FUNCTION_BLOCK "_UtilitiesFB"
{ S7_Optimized_Access := 'TRUE' }
VERSION : 0.1
   VAR_INPUT
      CPUSytemMemoryBits { ExternalAccessible := 'False'; ExternalVisible := 'False'; ExternalWritable := 'False'; } : Byte;   // Address of system memory byte
      CPUClockMemoryBits { ExternalAccessible := 'False'; ExternalVisible := 'False'; ExternalWritable := 'False'; } : Byte;   // Address of clock memory byte
      StartupDelaySP { ExternalAccessible := 'False'; ExternalVisible := 'False'; ExternalWritable := 'False'; } : Time;   // Delay before startup delay bit turned on
   END_VAR

   VAR
      AlwaysOn { ExternalAccessible := 'False'; ExternalVisible := 'False'; ExternalWritable := 'False'; } : Bool;   // Bit always TRUE
      AlwaysTrue { ExternalAccessible := 'False'; ExternalVisible := 'False'; ExternalWritable := 'False'; } : Bool;   // Bit always TRUE
      AlwaysOff { ExternalAccessible := 'False'; ExternalVisible := 'False'; ExternalWritable := 'False'; } : Bool;   // Bit always FALSE
      AlwaysFalse { ExternalAccessible := 'False'; ExternalVisible := 'False'; ExternalWritable := 'False'; } : Bool;   // Bit always FALSE
      FirstScan { ExternalAccessible := 'False'; ExternalVisible := 'False'; ExternalWritable := 'False'; } : Bool;   // Bit TRUE for only the first scan of the PLC
      StartupDelayDn { ExternalAccessible := 'False'; ExternalVisible := 'False'; ExternalWritable := 'False'; } : Bool;   // Bit initially FALSE, turning TRUE after preset delay
      StartupDelayTmr { ExternalAccessible := 'False'; ExternalVisible := 'False'; ExternalWritable := 'False'; OriginalPartName := 'IEC_TIMER'; LibVersion := '1.0'} : IEC_TIMER;
      Square_100ms { ExternalAccessible := 'False'; ExternalVisible := 'False'; ExternalWritable := 'False'; } : Bool;   // Bit FALSE/TRUE based on square wave (100 ms frequency)
      Square_100msONS { ExternalAccessible := 'False'; ExternalVisible := 'False'; ExternalWritable := 'False'; } : Bool;
      Pulse_100ms { ExternalAccessible := 'False'; ExternalVisible := 'False'; ExternalWritable := 'False'; } : Bool;   // Bit TRUE every 100 ms for one PLC scan
      Square_200ms { ExternalAccessible := 'False'; ExternalVisible := 'False'; ExternalWritable := 'False'; } : Bool;   // Bit FALSE/TRUE based on square wave (200 ms frequency)
      Square_200msONS { ExternalAccessible := 'False'; ExternalVisible := 'False'; ExternalWritable := 'False'; } : Bool;
      Pulse_200ms { ExternalAccessible := 'False'; ExternalVisible := 'False'; ExternalWritable := 'False'; } : Bool;   // Bit TRUE every 200 ms for one PLC scan
      Square_400ms { ExternalAccessible := 'False'; ExternalVisible := 'False'; ExternalWritable := 'False'; } : Bool;   // Bit FALSE/TRUE based on square wave (400 ms frequency)
      Square_400msONS { ExternalAccessible := 'False'; ExternalVisible := 'False'; ExternalWritable := 'False'; } : Bool;
      Pulse_400ms { ExternalAccessible := 'False'; ExternalVisible := 'False'; ExternalWritable := 'False'; } : Bool;   // Bit TRUE every 400 ms for one PLC scan
      Square_500ms { ExternalAccessible := 'False'; ExternalVisible := 'False'; ExternalWritable := 'False'; } : Bool;   // Bit FALSE/TRUE based on square wave (500 ms frequency)
      Square_500msONS { ExternalAccessible := 'False'; ExternalVisible := 'False'; ExternalWritable := 'False'; } : Bool;
      Pulse_500ms { ExternalAccessible := 'False'; ExternalVisible := 'False'; ExternalWritable := 'False'; } : Bool;   // Bit TRUE every 500 ms for one PLC scan
      Square_800ms { ExternalAccessible := 'False'; ExternalVisible := 'False'; ExternalWritable := 'False'; } : Bool;   // Bit FALSE/TRUE based on square wave (800 ms frequency)
      Square_800msONS { ExternalAccessible := 'False'; ExternalVisible := 'False'; ExternalWritable := 'False'; } : Bool;
      Pulse_800ms { ExternalAccessible := 'False'; ExternalVisible := 'False'; ExternalWritable := 'False'; } : Bool;   // Bit TRUE every 800 ms for one PLC scan
      Square_1s { ExternalAccessible := 'False'; ExternalVisible := 'False'; ExternalWritable := 'False'; } : Bool;   // Bit FALSE/TRUE based on square wave (1 s frequency)
      Square_1sONS { ExternalAccessible := 'False'; ExternalVisible := 'False'; ExternalWritable := 'False'; } : Bool;
      Pulse_1s { ExternalAccessible := 'False'; ExternalVisible := 'False'; ExternalWritable := 'False'; } : Bool;   // Bit TRUE every 1 s for one PLC scan
      Square_1600ms { ExternalAccessible := 'False'; ExternalVisible := 'False'; ExternalWritable := 'False'; } : Bool;   // Bit FALSE/TRUE based on square wave (1600 ms frequency)
      Square_1600msONS { ExternalAccessible := 'False'; ExternalVisible := 'False'; ExternalWritable := 'False'; } : Bool;
      Pulse_1600ms { ExternalAccessible := 'False'; ExternalVisible := 'False'; ExternalWritable := 'False'; } : Bool;   // Bit TRUE every 1600 ms for one PLC scan
      Square_2s { ExternalAccessible := 'False'; ExternalVisible := 'False'; ExternalWritable := 'False'; } : Bool;   // Bit FALSE/TRUE based on square wave (2 s frequency)
      Square_2sONS { ExternalAccessible := 'False'; ExternalVisible := 'False'; ExternalWritable := 'False'; } : Bool;
      Pulse_2s { ExternalAccessible := 'False'; ExternalVisible := 'False'; ExternalWritable := 'False'; } : Bool;   // Bit TRUE every 2 s for one PLC scan
      TestInProgress { ExternalAccessible := 'False'; ExternalVisible := 'False'; ExternalWritable := 'False'; } : Bool;   // Indicates which caller FC is used
      EPICS_Device_calls_precessed { ExternalAccessible := 'False'; ExternalVisible := 'False'; ExternalWritable := 'False'; } : Bool;   // Indicates which caller FC is used
   END_VAR

BEGIN
	//This block provides standard "Utilities" tags that can be used in the rest OF the PLC code such
	//as:
	//* Always On
	//* Always Off
	//* Startup Delay
	//* Pulses (different frequences)
	//* etc.

	//When using This block in your program, name the instance DB "Utilities" AND THEN you will be able TO use tags like "Utilities.AlwaysOn" in the rest OF your program.

	//This block relies On information provided BY the CPU. This needs TO be enabled in the CPU hardware configuration under System AND Clock Memory.
	//Enable both functions AND pick memory bytes you'd like TO use (defauls are %MB1 AND %MB0 respectively).
	//THEN connect the selected Byte TO the inputs OF This block.
	//

	//Bit TRUE for only the first scan of the PLC
	#FirstScan := #CPUSytemMemoryBits.%X0;

	//Bit always TRUE
	#AlwaysOn := #CPUSytemMemoryBits.%X2;
	#AlwaysTrue := #CPUSytemMemoryBits.%X2;

	//Bit always FALSE
	#AlwaysOff := #CPUSytemMemoryBits.%X3;
	#AlwaysFalse := #CPUSytemMemoryBits.%X3;

	//Bit initially FALSE, turning TRUE after preset delay
	#StartupDelayTmr.TON(IN := #AlwaysTrue,
	                     PT := #StartupDelaySP,
	                     Q => #StartupDelayDn);

	//Bit TRUE every 100 ms FOR one PLC scan
	#Square_100ms := #CPUClockMemoryBits.%X0;
	"UTIL_P_TRIG"("i_Input Bit" := #Square_100ms,
	              "iq_Trigger Bit" := #Square_100msONS,
	              "iq_Pulse Bit" := #Pulse_100ms);

	//Bit TRUE every 200 ms FOR one PLC scan
	#Square_200ms := #CPUClockMemoryBits.%X1;
	"UTIL_P_TRIG"("i_Input Bit" := #Square_200ms,
	              "iq_Trigger Bit" := #Square_200msONS,
	              "iq_Pulse Bit" := #Pulse_200ms);

	//Bit TRUE every 400 ms FOR one PLC scan
	#Square_400ms := #CPUClockMemoryBits.%X2;
	"UTIL_P_TRIG"("i_Input Bit" := #Square_400ms,
	              "iq_Trigger Bit" := #Square_400msONS,
	              "iq_Pulse Bit" := #Pulse_400ms);

	//Bit TRUE every 500 ms FOR one PLC scan
	#Square_500ms := #CPUClockMemoryBits.%X3;
	"UTIL_P_TRIG"("i_Input Bit" := #Square_500ms,
	              "iq_Trigger Bit" := #Square_500msONS,
	              "iq_Pulse Bit" := #Pulse_500ms);

	//Bit TRUE every 800 ms FOR one PLC scan
	#Square_800ms := #CPUClockMemoryBits.%X4;
	"UTIL_P_TRIG"("i_Input Bit" := #Square_800ms,
	              "iq_Trigger Bit" := #Square_800msONS,
	              "iq_Pulse Bit" := #Pulse_800ms);

	//Bit TRUE every 1 s FOR one PLC scan
	#Square_1s := #CPUClockMemoryBits.%X5;
	"UTIL_P_TRIG"("i_Input Bit" := #Square_1s,
	              "iq_Trigger Bit" := #Square_1sONS,
	              "iq_Pulse Bit" := #Pulse_1s);

	//Bit TRUE every 1600 ms FOR one PLC scan
	#Square_1600ms := #CPUClockMemoryBits.%X6;
	"UTIL_P_TRIG"("i_Input Bit" := #Square_1600ms,
	              "iq_Trigger Bit" := #Square_1600msONS,
	              "iq_Pulse Bit" := #Pulse_1600ms);

	//Bit TRUE every 2s FOR one PLC scan
	#Square_2s := #CPUClockMemoryBits.%X7;
	"UTIL_P_TRIG"("i_Input Bit" := #Square_2s,
	              "iq_Trigger Bit" := #Square_2sONS,
	              "iq_Pulse Bit" := #Pulse_2s);

END_FUNCTION_BLOCK
DATA_BLOCK "Utilities"
{ S7_Optimized_Access := 'TRUE' }
VERSION : 0.1
NON_RETAIN
"_UtilitiesFB"

BEGIN

END_DATA_BLOCK
FUNCTION_BLOCK "DEVTYPE_ISRC_LEBT_BDump"
{ S7_Optimized_Access := 'TRUE' }
VERSION : 1.0
   VAR_INPUT
      "WtrFlowOK" { ExternalAccessible := 'True'; ExternalVisible := 'False'; ExternalWritable := 'False'; } : BOOL;   //EPICS Status variable: WtrFlowOK
   EPICSToPLCLength { ExternalAccessible := 'False'; ExternalVisible := 'False'; ExternalWritable := 'False'; } : Int;   // Length of device command register array (in words)
   EPICSToPLCDataBlockOffset { ExternalAccessible := 'False'; ExternalVisible := 'False'; ExternalWritable := 'False'; } : Int;   // Offset in EPICS->PLC comms block where this device data resides (in words)
   EPICSToPLCParametersStart { ExternalAccessible := 'False'; ExternalVisible := 'False'; ExternalWritable := 'False'; } : Int;   // The border offset between the Command and the Parameter area
   PLCToEPICSLength { ExternalAccessible := 'False'; ExternalVisible := 'False'; ExternalWritable := 'False'; } : Int;   // Length of device status register array (in words)
   PLCToEPICSDataBlockOffset { ExternalAccessible := 'False'; ExternalVisible := 'False'; ExternalWritable := 'False'; } : Int;   // Offset in PLC->EPICS comms block where this device data resides (in words)
   END_VAR
   VAR_OUTPUT
      DEVICE_PARAM_OK { ExternalAccessible := 'False'; ExternalVisible := 'False'; ExternalWritable := 'False'; } : Bool;
   END_VAR
   VAR_IN_OUT
   END_VAR
   Var DB_SPECIFIC
      MyWord { ExternalAccessible := 'False'; ExternalVisible := 'False'; ExternalWritable := 'False'; } : Word;
      MyBytesinWord { ExternalAccessible := 'False'; ExternalVisible := 'False'; ExternalWritable := 'False'; } AT MyWord : Array[0..1] of Byte;
      MyBoolsinWord { ExternalAccessible := 'False'; ExternalVisible := 'False'; ExternalWritable := 'False'; } AT MyWord : Array[0..15] of Bool;
      MyDInt { ExternalAccessible := 'False'; ExternalVisible := 'False'; ExternalWritable := 'False'; } : DInt;
      MyWordsinDint { ExternalAccessible := 'False'; ExternalVisible := 'False'; ExternalWritable := 'False'; } AT MyDInt : Array[0..1] of Word;
      MyReal { ExternalAccessible := 'False'; ExternalVisible := 'False'; ExternalWritable := 'False'; } : Real;
      MyWordsinReal { ExternalAccessible := 'False'; ExternalVisible := 'False'; ExternalWritable := 'False'; } AT MyReal : Array[0..1] of Word;
      MyInt { ExternalAccessible := 'False'; ExternalVisible := 'False'; ExternalWritable := 'False'; } : Int;
      MyWordinInt { ExternalAccessible := 'False'; ExternalVisible := 'False'; ExternalWritable := 'False'; } AT MyInt : Word;
      MyDWord { ExternalAccessible := 'False'; ExternalVisible := 'False'; ExternalWritable := 'False'; } : DWord;
      MyWordsinDWord { ExternalAccessible := 'False'; ExternalVisible := 'False'; ExternalWritable := 'False'; } AT MyDWord : Array[0..1] of Word;
      MyTime { ExternalAccessible := 'False'; ExternalVisible := 'False'; ExternalWritable := 'False'; } : Time;
      MyWordsinTime { ExternalAccessible := 'False'; ExternalVisible := 'False'; ExternalWritable := 'False'; } AT MyTime : Array[0..1] of Word;
      MyString { ExternalAccessible := 'False'; ExternalVisible := 'False'; ExternalWritable := 'False'; } : String[40];
      MyWordsinString { ExternalAccessible := 'False'; ExternalVisible := 'False'; ExternalWritable := 'False'; } AT MyString : Array[0..20] of Word;
   END_VAR
   VAR_TEMP
      HashModbus : DInt;
      HashIFA : DInt;
      HashTIAMap : DInt;
      i : Int;
   END_VAR
    //Author: Miklos Boros (miklos.boros@esss.se), Copyrigth 2017-2019 by European Spallation Source, Lund
    //This block was generated by PLCFactory, please don't change it MANUALLY!
    //Input File Name: ISrc-010_Ctrl-PLC-01-template-IFA-20191106135317.ifa
    //Generated: 20191106135317
    //According to HASH: 1347332123
    //Device type: ISRC_LEBT_BDump
    //Description: This function does the variable mapping for a device. All device-variable will be linked to an interface variable defined in this block.

    //********************************************
    //****************HASH check******************
    //********************************************


    #MyWordsinDint[0] := "EPICSToPLC"."Word"[0];
    #MyWordsinDint[1] := "EPICSToPLC"."Word"[1];
    #HashModbus := #MyDInt; //Hash from EPICS/ModbusTCP

    #HashIFA := 1347332123; //Hash from Interface Factory as a constant

    #MyWordsinDint[0] := "PLCToEPICS"."Word"[0];
    #MyWordsinDint[1] := "PLCToEPICS"."Word"[1];
    #HashTIAMap := #MyDInt; //Hash from PLCFactory TIA Map


    IF ((#HashIFA = #HashModbus) AND (#HashModbus = #HashTIAMap)) THEN //Check CRCs
        #DEVICE_PARAM_OK := TRUE;
       //###########################  LEBT Beam Dump  ##############################
       //###########################
       //STATUS BLOCK
       //###########################

    //********************************************
    //*************STATUS VARIABLES***************
    //********************************************


       #MyWord := W#0;
       #MyBoolsinWord[8] := #"WtrFlowOK";    //EPICSName: WtrFlowOK
       "PLCToEPICS"."Word"[#PLCToEPICSDataBlockOffset + 0] := #MyWord;
    Else
       #DEVICE_PARAM_OK := FALSE; //Invalid Hash
    END_IF;
END_FUNCTION_BLOCK
FUNCTION_BLOCK "DEVTYPE_ISRC_LEBT_CHOP"
{ S7_Optimized_Access := 'TRUE' }
VERSION : 1.0
   VAR_INPUT
      "PwrSysOK" { ExternalAccessible := 'True'; ExternalVisible := 'False'; ExternalWritable := 'False'; } : BOOL;   //EPICS Status variable: PwrSysOK
      "ChopVoltAlarmR" { ExternalAccessible := 'True'; ExternalVisible := 'False'; ExternalWritable := 'False'; } : BOOL;   //EPICS Status variable: ChopVoltAlarmR
      "WtrFlowOK" { ExternalAccessible := 'True'; ExternalVisible := 'False'; ExternalWritable := 'False'; } : BOOL;   //EPICS Status variable: WtrFlowOK
      "HVEnCmdRB" { ExternalAccessible := 'True'; ExternalVisible := 'False'; ExternalWritable := 'False'; } : BOOL;   //EPICS Status variable: HVEnCmdRB
   EPICSToPLCLength { ExternalAccessible := 'False'; ExternalVisible := 'False'; ExternalWritable := 'False'; } : Int;   // Length of device command register array (in words)
   EPICSToPLCDataBlockOffset { ExternalAccessible := 'False'; ExternalVisible := 'False'; ExternalWritable := 'False'; } : Int;   // Offset in EPICS->PLC comms block where this device data resides (in words)
   EPICSToPLCParametersStart { ExternalAccessible := 'False'; ExternalVisible := 'False'; ExternalWritable := 'False'; } : Int;   // The border offset between the Command and the Parameter area
   PLCToEPICSLength { ExternalAccessible := 'False'; ExternalVisible := 'False'; ExternalWritable := 'False'; } : Int;   // Length of device status register array (in words)
   PLCToEPICSDataBlockOffset { ExternalAccessible := 'False'; ExternalVisible := 'False'; ExternalWritable := 'False'; } : Int;   // Offset in PLC->EPICS comms block where this device data resides (in words)
   END_VAR
   VAR_OUTPUT
      "HVEnOnCmd" { ExternalAccessible := 'True'; ExternalVisible := 'False'; ExternalWritable := 'False'; } : BOOL;   //EPICS Command variable: HVEnOnCmd
      "HVEnOffCmd" { ExternalAccessible := 'True'; ExternalVisible := 'False'; ExternalWritable := 'False'; } : BOOL;   //EPICS Command variable: HVEnOffCmd
      DEVICE_PARAM_OK { ExternalAccessible := 'False'; ExternalVisible := 'False'; ExternalWritable := 'False'; } : Bool;
   END_VAR
   VAR_IN_OUT
   END_VAR
   Var DB_SPECIFIC
      MyWord { ExternalAccessible := 'False'; ExternalVisible := 'False'; ExternalWritable := 'False'; } : Word;
      MyBytesinWord { ExternalAccessible := 'False'; ExternalVisible := 'False'; ExternalWritable := 'False'; } AT MyWord : Array[0..1] of Byte;
      MyBoolsinWord { ExternalAccessible := 'False'; ExternalVisible := 'False'; ExternalWritable := 'False'; } AT MyWord : Array[0..15] of Bool;
      MyDInt { ExternalAccessible := 'False'; ExternalVisible := 'False'; ExternalWritable := 'False'; } : DInt;
      MyWordsinDint { ExternalAccessible := 'False'; ExternalVisible := 'False'; ExternalWritable := 'False'; } AT MyDInt : Array[0..1] of Word;
      MyReal { ExternalAccessible := 'False'; ExternalVisible := 'False'; ExternalWritable := 'False'; } : Real;
      MyWordsinReal { ExternalAccessible := 'False'; ExternalVisible := 'False'; ExternalWritable := 'False'; } AT MyReal : Array[0..1] of Word;
      MyInt { ExternalAccessible := 'False'; ExternalVisible := 'False'; ExternalWritable := 'False'; } : Int;
      MyWordinInt { ExternalAccessible := 'False'; ExternalVisible := 'False'; ExternalWritable := 'False'; } AT MyInt : Word;
      MyDWord { ExternalAccessible := 'False'; ExternalVisible := 'False'; ExternalWritable := 'False'; } : DWord;
      MyWordsinDWord { ExternalAccessible := 'False'; ExternalVisible := 'False'; ExternalWritable := 'False'; } AT MyDWord : Array[0..1] of Word;
      MyTime { ExternalAccessible := 'False'; ExternalVisible := 'False'; ExternalWritable := 'False'; } : Time;
      MyWordsinTime { ExternalAccessible := 'False'; ExternalVisible := 'False'; ExternalWritable := 'False'; } AT MyTime : Array[0..1] of Word;
      MyString { ExternalAccessible := 'False'; ExternalVisible := 'False'; ExternalWritable := 'False'; } : String[40];
      MyWordsinString { ExternalAccessible := 'False'; ExternalVisible := 'False'; ExternalWritable := 'False'; } AT MyString : Array[0..20] of Word;
   END_VAR
   VAR_TEMP
      HashModbus : DInt;
      HashIFA : DInt;
      HashTIAMap : DInt;
      i : Int;
   END_VAR
    //Author: Miklos Boros (miklos.boros@esss.se), Copyrigth 2017-2019 by European Spallation Source, Lund
    //This block was generated by PLCFactory, please don't change it MANUALLY!
    //Input File Name: ISrc-010_Ctrl-PLC-01-template-IFA-20191106135317.ifa
    //Generated: 20191106135317
    //According to HASH: 1347332123
    //Device type: ISRC_LEBT_CHOP
    //Description: This function does the variable mapping for a device. All device-variable will be linked to an interface variable defined in this block.

    //********************************************
    //****************HASH check******************
    //********************************************


    #MyWordsinDint[0] := "EPICSToPLC"."Word"[0];
    #MyWordsinDint[1] := "EPICSToPLC"."Word"[1];
    #HashModbus := #MyDInt; //Hash from EPICS/ModbusTCP

    #HashIFA := 1347332123; //Hash from Interface Factory as a constant

    #MyWordsinDint[0] := "PLCToEPICS"."Word"[0];
    #MyWordsinDint[1] := "PLCToEPICS"."Word"[1];
    #HashTIAMap := #MyDInt; //Hash from PLCFactory TIA Map


    IF ((#HashIFA = #HashModbus) AND (#HashModbus = #HashTIAMap)) THEN //Check CRCs
        #DEVICE_PARAM_OK := TRUE;
       //###########################  LEBT Chopper  ##############################
       //###########################
       //STATUS BLOCK
       //###########################

    //********************************************
    //*************STATUS VARIABLES***************
    //********************************************


       #MyWord := W#0;
       #MyBoolsinWord[8] := #"PwrSysOK";    //EPICSName: PwrSysOK
       #MyBoolsinWord[9] := #"ChopVoltAlarmR";    //EPICSName: ChopVoltAlarmR
       #MyBoolsinWord[10] := #"WtrFlowOK";    //EPICSName: WtrFlowOK
       #MyBoolsinWord[11] := #"HVEnCmdRB";    //EPICSName: HVEnCmdRB
       "PLCToEPICS"."Word"[#PLCToEPICSDataBlockOffset + 0] := #MyWord;

    //********************************************
    //*************COMMAND VARIABLES**************
    //********************************************


       #MyWord := "EPICSToPLC"."Word"[#EPICSToPLCDataBlockOffset + 0];
       IF (NOT "Utilities".TestInProgress) THEN
       	"EPICSToPLC"."Word"[#EPICSToPLCDataBlockOffset + 0] := 0;
       END_IF;
       #"HVEnOnCmd" := #MyBoolsinWord[8];    //EPICSName: HVEnOnCmd
       #"HVEnOffCmd" := #MyBoolsinWord[9];    //EPICSName: HVEnOffCmd
    Else
       #DEVICE_PARAM_OK := FALSE; //Invalid Hash
    END_IF;
END_FUNCTION_BLOCK
FUNCTION_BLOCK "DEVTYPE_ISRC_LEBT_COIL_SOLENOID"
{ S7_Optimized_Access := 'TRUE' }
VERSION : 1.0
   VAR_INPUT
      "WtrFlowOK" { ExternalAccessible := 'True'; ExternalVisible := 'False'; ExternalWritable := 'False'; } : BOOL;   //EPICS Status variable: WtrFlowOK
      "WtrTempOK" { ExternalAccessible := 'True'; ExternalVisible := 'False'; ExternalWritable := 'False'; } : BOOL;   //EPICS Status variable: WtrTempOK
   EPICSToPLCLength { ExternalAccessible := 'False'; ExternalVisible := 'False'; ExternalWritable := 'False'; } : Int;   // Length of device command register array (in words)
   EPICSToPLCDataBlockOffset { ExternalAccessible := 'False'; ExternalVisible := 'False'; ExternalWritable := 'False'; } : Int;   // Offset in EPICS->PLC comms block where this device data resides (in words)
   EPICSToPLCParametersStart { ExternalAccessible := 'False'; ExternalVisible := 'False'; ExternalWritable := 'False'; } : Int;   // The border offset between the Command and the Parameter area
   PLCToEPICSLength { ExternalAccessible := 'False'; ExternalVisible := 'False'; ExternalWritable := 'False'; } : Int;   // Length of device status register array (in words)
   PLCToEPICSDataBlockOffset { ExternalAccessible := 'False'; ExternalVisible := 'False'; ExternalWritable := 'False'; } : Int;   // Offset in PLC->EPICS comms block where this device data resides (in words)
   END_VAR
   VAR_OUTPUT
      DEVICE_PARAM_OK { ExternalAccessible := 'False'; ExternalVisible := 'False'; ExternalWritable := 'False'; } : Bool;
   END_VAR
   VAR_IN_OUT
   END_VAR
   Var DB_SPECIFIC
      MyWord { ExternalAccessible := 'False'; ExternalVisible := 'False'; ExternalWritable := 'False'; } : Word;
      MyBytesinWord { ExternalAccessible := 'False'; ExternalVisible := 'False'; ExternalWritable := 'False'; } AT MyWord : Array[0..1] of Byte;
      MyBoolsinWord { ExternalAccessible := 'False'; ExternalVisible := 'False'; ExternalWritable := 'False'; } AT MyWord : Array[0..15] of Bool;
      MyDInt { ExternalAccessible := 'False'; ExternalVisible := 'False'; ExternalWritable := 'False'; } : DInt;
      MyWordsinDint { ExternalAccessible := 'False'; ExternalVisible := 'False'; ExternalWritable := 'False'; } AT MyDInt : Array[0..1] of Word;
      MyReal { ExternalAccessible := 'False'; ExternalVisible := 'False'; ExternalWritable := 'False'; } : Real;
      MyWordsinReal { ExternalAccessible := 'False'; ExternalVisible := 'False'; ExternalWritable := 'False'; } AT MyReal : Array[0..1] of Word;
      MyInt { ExternalAccessible := 'False'; ExternalVisible := 'False'; ExternalWritable := 'False'; } : Int;
      MyWordinInt { ExternalAccessible := 'False'; ExternalVisible := 'False'; ExternalWritable := 'False'; } AT MyInt : Word;
      MyDWord { ExternalAccessible := 'False'; ExternalVisible := 'False'; ExternalWritable := 'False'; } : DWord;
      MyWordsinDWord { ExternalAccessible := 'False'; ExternalVisible := 'False'; ExternalWritable := 'False'; } AT MyDWord : Array[0..1] of Word;
      MyTime { ExternalAccessible := 'False'; ExternalVisible := 'False'; ExternalWritable := 'False'; } : Time;
      MyWordsinTime { ExternalAccessible := 'False'; ExternalVisible := 'False'; ExternalWritable := 'False'; } AT MyTime : Array[0..1] of Word;
      MyString { ExternalAccessible := 'False'; ExternalVisible := 'False'; ExternalWritable := 'False'; } : String[40];
      MyWordsinString { ExternalAccessible := 'False'; ExternalVisible := 'False'; ExternalWritable := 'False'; } AT MyString : Array[0..20] of Word;
   END_VAR
   VAR_TEMP
      HashModbus : DInt;
      HashIFA : DInt;
      HashTIAMap : DInt;
      i : Int;
   END_VAR
    //Author: Miklos Boros (miklos.boros@esss.se), Copyrigth 2017-2019 by European Spallation Source, Lund
    //This block was generated by PLCFactory, please don't change it MANUALLY!
    //Input File Name: ISrc-010_Ctrl-PLC-01-template-IFA-20191106135317.ifa
    //Generated: 20191106135317
    //According to HASH: 1347332123
    //Device type: ISRC_LEBT_COIL_SOLENOID
    //Description: This function does the variable mapping for a device. All device-variable will be linked to an interface variable defined in this block.

    //********************************************
    //****************HASH check******************
    //********************************************


    #MyWordsinDint[0] := "EPICSToPLC"."Word"[0];
    #MyWordsinDint[1] := "EPICSToPLC"."Word"[1];
    #HashModbus := #MyDInt; //Hash from EPICS/ModbusTCP

    #HashIFA := 1347332123; //Hash from Interface Factory as a constant

    #MyWordsinDint[0] := "PLCToEPICS"."Word"[0];
    #MyWordsinDint[1] := "PLCToEPICS"."Word"[1];
    #HashTIAMap := #MyDInt; //Hash from PLCFactory TIA Map


    IF ((#HashIFA = #HashModbus) AND (#HashModbus = #HashTIAMap)) THEN //Check CRCs
        #DEVICE_PARAM_OK := TRUE;
       //###########################  ISRC_LEBT Coils and Solenoids Water Flow and Temperature Status  ##############################
       //###########################
       //STATUS BLOCK
       //###########################

    //********************************************
    //*************STATUS VARIABLES***************
    //********************************************


       #MyWord := W#0;
       #MyBoolsinWord[8] := #"WtrFlowOK";    //EPICSName: WtrFlowOK
       #MyBoolsinWord[9] := #"WtrTempOK";    //EPICSName: WtrTempOK
       "PLCToEPICS"."Word"[#PLCToEPICSDataBlockOffset + 0] := #MyWord;
    Else
       #DEVICE_PARAM_OK := FALSE; //Invalid Hash
    END_IF;
END_FUNCTION_BLOCK
FUNCTION_BLOCK "DEVTYPE_ISRC_LEBT_COLL"
{ S7_Optimized_Access := 'TRUE' }
VERSION : 1.0
   VAR_INPUT
      "WtrFlowOK" { ExternalAccessible := 'True'; ExternalVisible := 'False'; ExternalWritable := 'False'; } : BOOL;   //EPICS Status variable: WtrFlowOK
   EPICSToPLCLength { ExternalAccessible := 'False'; ExternalVisible := 'False'; ExternalWritable := 'False'; } : Int;   // Length of device command register array (in words)
   EPICSToPLCDataBlockOffset { ExternalAccessible := 'False'; ExternalVisible := 'False'; ExternalWritable := 'False'; } : Int;   // Offset in EPICS->PLC comms block where this device data resides (in words)
   EPICSToPLCParametersStart { ExternalAccessible := 'False'; ExternalVisible := 'False'; ExternalWritable := 'False'; } : Int;   // The border offset between the Command and the Parameter area
   PLCToEPICSLength { ExternalAccessible := 'False'; ExternalVisible := 'False'; ExternalWritable := 'False'; } : Int;   // Length of device status register array (in words)
   PLCToEPICSDataBlockOffset { ExternalAccessible := 'False'; ExternalVisible := 'False'; ExternalWritable := 'False'; } : Int;   // Offset in PLC->EPICS comms block where this device data resides (in words)
   END_VAR
   VAR_OUTPUT
      DEVICE_PARAM_OK { ExternalAccessible := 'False'; ExternalVisible := 'False'; ExternalWritable := 'False'; } : Bool;
   END_VAR
   VAR_IN_OUT
   END_VAR
   Var DB_SPECIFIC
      MyWord { ExternalAccessible := 'False'; ExternalVisible := 'False'; ExternalWritable := 'False'; } : Word;
      MyBytesinWord { ExternalAccessible := 'False'; ExternalVisible := 'False'; ExternalWritable := 'False'; } AT MyWord : Array[0..1] of Byte;
      MyBoolsinWord { ExternalAccessible := 'False'; ExternalVisible := 'False'; ExternalWritable := 'False'; } AT MyWord : Array[0..15] of Bool;
      MyDInt { ExternalAccessible := 'False'; ExternalVisible := 'False'; ExternalWritable := 'False'; } : DInt;
      MyWordsinDint { ExternalAccessible := 'False'; ExternalVisible := 'False'; ExternalWritable := 'False'; } AT MyDInt : Array[0..1] of Word;
      MyReal { ExternalAccessible := 'False'; ExternalVisible := 'False'; ExternalWritable := 'False'; } : Real;
      MyWordsinReal { ExternalAccessible := 'False'; ExternalVisible := 'False'; ExternalWritable := 'False'; } AT MyReal : Array[0..1] of Word;
      MyInt { ExternalAccessible := 'False'; ExternalVisible := 'False'; ExternalWritable := 'False'; } : Int;
      MyWordinInt { ExternalAccessible := 'False'; ExternalVisible := 'False'; ExternalWritable := 'False'; } AT MyInt : Word;
      MyDWord { ExternalAccessible := 'False'; ExternalVisible := 'False'; ExternalWritable := 'False'; } : DWord;
      MyWordsinDWord { ExternalAccessible := 'False'; ExternalVisible := 'False'; ExternalWritable := 'False'; } AT MyDWord : Array[0..1] of Word;
      MyTime { ExternalAccessible := 'False'; ExternalVisible := 'False'; ExternalWritable := 'False'; } : Time;
      MyWordsinTime { ExternalAccessible := 'False'; ExternalVisible := 'False'; ExternalWritable := 'False'; } AT MyTime : Array[0..1] of Word;
      MyString { ExternalAccessible := 'False'; ExternalVisible := 'False'; ExternalWritable := 'False'; } : String[40];
      MyWordsinString { ExternalAccessible := 'False'; ExternalVisible := 'False'; ExternalWritable := 'False'; } AT MyString : Array[0..20] of Word;
   END_VAR
   VAR_TEMP
      HashModbus : DInt;
      HashIFA : DInt;
      HashTIAMap : DInt;
      i : Int;
   END_VAR
    //Author: Miklos Boros (miklos.boros@esss.se), Copyrigth 2017-2019 by European Spallation Source, Lund
    //This block was generated by PLCFactory, please don't change it MANUALLY!
    //Input File Name: ISrc-010_Ctrl-PLC-01-template-IFA-20191106135317.ifa
    //Generated: 20191106135317
    //According to HASH: 1347332123
    //Device type: ISRC_LEBT_COLL
    //Description: This function does the variable mapping for a device. All device-variable will be linked to an interface variable defined in this block.

    //********************************************
    //****************HASH check******************
    //********************************************


    #MyWordsinDint[0] := "EPICSToPLC"."Word"[0];
    #MyWordsinDint[1] := "EPICSToPLC"."Word"[1];
    #HashModbus := #MyDInt; //Hash from EPICS/ModbusTCP

    #HashIFA := 1347332123; //Hash from Interface Factory as a constant

    #MyWordsinDint[0] := "PLCToEPICS"."Word"[0];
    #MyWordsinDint[1] := "PLCToEPICS"."Word"[1];
    #HashTIAMap := #MyDInt; //Hash from PLCFactory TIA Map


    IF ((#HashIFA = #HashModbus) AND (#HashModbus = #HashTIAMap)) THEN //Check CRCs
        #DEVICE_PARAM_OK := TRUE;
       //###########################  LEBT Collimator  ##############################
       //###########################
       //STATUS BLOCK
       //###########################

    //********************************************
    //*************STATUS VARIABLES***************
    //********************************************


       #MyWord := W#0;
       #MyBoolsinWord[8] := #"WtrFlowOK";    //EPICSName: WtrFlowOK
       "PLCToEPICS"."Word"[#PLCToEPICSDataBlockOffset + 0] := #MyWord;
    Else
       #DEVICE_PARAM_OK := FALSE; //Invalid Hash
    END_IF;
END_FUNCTION_BLOCK
FUNCTION_BLOCK "DEVTYPE_ISRC_LEBT_HVIT"
{ S7_Optimized_Access := 'TRUE' }
VERSION : 1.0
   VAR_INPUT
      "LidOpenR" { ExternalAccessible := 'True'; ExternalVisible := 'False'; ExternalWritable := 'False'; } : BOOL;   //EPICS Status variable: LidOpenR
      "OilTempOK" { ExternalAccessible := 'True'; ExternalVisible := 'False'; ExternalWritable := 'False'; } : BOOL;   //EPICS Status variable: OilTempOK
   EPICSToPLCLength { ExternalAccessible := 'False'; ExternalVisible := 'False'; ExternalWritable := 'False'; } : Int;   // Length of device command register array (in words)
   EPICSToPLCDataBlockOffset { ExternalAccessible := 'False'; ExternalVisible := 'False'; ExternalWritable := 'False'; } : Int;   // Offset in EPICS->PLC comms block where this device data resides (in words)
   EPICSToPLCParametersStart { ExternalAccessible := 'False'; ExternalVisible := 'False'; ExternalWritable := 'False'; } : Int;   // The border offset between the Command and the Parameter area
   PLCToEPICSLength { ExternalAccessible := 'False'; ExternalVisible := 'False'; ExternalWritable := 'False'; } : Int;   // Length of device status register array (in words)
   PLCToEPICSDataBlockOffset { ExternalAccessible := 'False'; ExternalVisible := 'False'; ExternalWritable := 'False'; } : Int;   // Offset in PLC->EPICS comms block where this device data resides (in words)
   END_VAR
   VAR_OUTPUT
      DEVICE_PARAM_OK { ExternalAccessible := 'False'; ExternalVisible := 'False'; ExternalWritable := 'False'; } : Bool;
   END_VAR
   VAR_IN_OUT
   END_VAR
   Var DB_SPECIFIC
      MyWord { ExternalAccessible := 'False'; ExternalVisible := 'False'; ExternalWritable := 'False'; } : Word;
      MyBytesinWord { ExternalAccessible := 'False'; ExternalVisible := 'False'; ExternalWritable := 'False'; } AT MyWord : Array[0..1] of Byte;
      MyBoolsinWord { ExternalAccessible := 'False'; ExternalVisible := 'False'; ExternalWritable := 'False'; } AT MyWord : Array[0..15] of Bool;
      MyDInt { ExternalAccessible := 'False'; ExternalVisible := 'False'; ExternalWritable := 'False'; } : DInt;
      MyWordsinDint { ExternalAccessible := 'False'; ExternalVisible := 'False'; ExternalWritable := 'False'; } AT MyDInt : Array[0..1] of Word;
      MyReal { ExternalAccessible := 'False'; ExternalVisible := 'False'; ExternalWritable := 'False'; } : Real;
      MyWordsinReal { ExternalAccessible := 'False'; ExternalVisible := 'False'; ExternalWritable := 'False'; } AT MyReal : Array[0..1] of Word;
      MyInt { ExternalAccessible := 'False'; ExternalVisible := 'False'; ExternalWritable := 'False'; } : Int;
      MyWordinInt { ExternalAccessible := 'False'; ExternalVisible := 'False'; ExternalWritable := 'False'; } AT MyInt : Word;
      MyDWord { ExternalAccessible := 'False'; ExternalVisible := 'False'; ExternalWritable := 'False'; } : DWord;
      MyWordsinDWord { ExternalAccessible := 'False'; ExternalVisible := 'False'; ExternalWritable := 'False'; } AT MyDWord : Array[0..1] of Word;
      MyTime { ExternalAccessible := 'False'; ExternalVisible := 'False'; ExternalWritable := 'False'; } : Time;
      MyWordsinTime { ExternalAccessible := 'False'; ExternalVisible := 'False'; ExternalWritable := 'False'; } AT MyTime : Array[0..1] of Word;
      MyString { ExternalAccessible := 'False'; ExternalVisible := 'False'; ExternalWritable := 'False'; } : String[40];
      MyWordsinString { ExternalAccessible := 'False'; ExternalVisible := 'False'; ExternalWritable := 'False'; } AT MyString : Array[0..20] of Word;
   END_VAR
   VAR_TEMP
      HashModbus : DInt;
      HashIFA : DInt;
      HashTIAMap : DInt;
      i : Int;
   END_VAR
    //Author: Miklos Boros (miklos.boros@esss.se), Copyrigth 2017-2019 by European Spallation Source, Lund
    //This block was generated by PLCFactory, please don't change it MANUALLY!
    //Input File Name: ISrc-010_Ctrl-PLC-01-template-IFA-20191106135317.ifa
    //Generated: 20191106135317
    //According to HASH: 1347332123
    //Device type: ISRC_LEBT_HVIT
    //Description: This function does the variable mapping for a device. All device-variable will be linked to an interface variable defined in this block.

    //********************************************
    //****************HASH check******************
    //********************************************


    #MyWordsinDint[0] := "EPICSToPLC"."Word"[0];
    #MyWordsinDint[1] := "EPICSToPLC"."Word"[1];
    #HashModbus := #MyDInt; //Hash from EPICS/ModbusTCP

    #HashIFA := 1347332123; //Hash from Interface Factory as a constant

    #MyWordsinDint[0] := "PLCToEPICS"."Word"[0];
    #MyWordsinDint[1] := "PLCToEPICS"."Word"[1];
    #HashTIAMap := #MyDInt; //Hash from PLCFactory TIA Map


    IF ((#HashIFA = #HashModbus) AND (#HashModbus = #HashTIAMap)) THEN //Check CRCs
        #DEVICE_PARAM_OK := TRUE;
       //###########################  ISRC HV Isolation Transformer  ##############################
       //###########################
       //STATUS BLOCK
       //###########################

    //********************************************
    //*************STATUS VARIABLES***************
    //********************************************


       #MyWord := W#0;
       #MyBoolsinWord[8] := #"LidOpenR";    //EPICSName: LidOpenR
       #MyBoolsinWord[9] := #"OilTempOK";    //EPICSName: OilTempOK
       "PLCToEPICS"."Word"[#PLCToEPICSDataBlockOffset + 0] := #MyWord;
    Else
       #DEVICE_PARAM_OK := FALSE; //Invalid Hash
    END_IF;
END_FUNCTION_BLOCK
FUNCTION_BLOCK "DEVTYPE_ISRC_LEBT_HVPS"
{ S7_Optimized_Access := 'TRUE' }
VERSION : 1.0
   VAR_INPUT
      "ITLckEnCmdR" { ExternalAccessible := 'True'; ExternalVisible := 'False'; ExternalWritable := 'False'; } : BOOL;   //EPICS Status variable: ITLckEnCmdR
      "HVPSVolOK_Magtr" { ExternalAccessible := 'True'; ExternalVisible := 'False'; ExternalWritable := 'False'; } : BOOL;   //EPICS Status variable: HVPSVolOK_Magtr
   EPICSToPLCLength { ExternalAccessible := 'False'; ExternalVisible := 'False'; ExternalWritable := 'False'; } : Int;   // Length of device command register array (in words)
   EPICSToPLCDataBlockOffset { ExternalAccessible := 'False'; ExternalVisible := 'False'; ExternalWritable := 'False'; } : Int;   // Offset in EPICS->PLC comms block where this device data resides (in words)
   EPICSToPLCParametersStart { ExternalAccessible := 'False'; ExternalVisible := 'False'; ExternalWritable := 'False'; } : Int;   // The border offset between the Command and the Parameter area
   PLCToEPICSLength { ExternalAccessible := 'False'; ExternalVisible := 'False'; ExternalWritable := 'False'; } : Int;   // Length of device status register array (in words)
   PLCToEPICSDataBlockOffset { ExternalAccessible := 'False'; ExternalVisible := 'False'; ExternalWritable := 'False'; } : Int;   // Offset in PLC->EPICS comms block where this device data resides (in words)
   END_VAR
   VAR_OUTPUT
      "ESTOP" { ExternalAccessible := 'True'; ExternalVisible := 'False'; ExternalWritable := 'False'; } : BOOL;   //EPICS Command variable: ESTOP
      "iVolR" { ExternalAccessible := 'True'; ExternalVisible := 'False'; ExternalWritable := 'False'; } : REAL;   //EPICS Parameter variable: iVolR
      "EPICSConnErr" { ExternalAccessible := 'True'; ExternalVisible := 'False'; ExternalWritable := 'False'; } : BOOL;   //EPICS Parameter variable: EPICSConnErr
      DEVICE_PARAM_OK { ExternalAccessible := 'False'; ExternalVisible := 'False'; ExternalWritable := 'False'; } : Bool;
   END_VAR
   VAR_IN_OUT
   END_VAR
   Var DB_SPECIFIC
      MyWord { ExternalAccessible := 'False'; ExternalVisible := 'False'; ExternalWritable := 'False'; } : Word;
      MyBytesinWord { ExternalAccessible := 'False'; ExternalVisible := 'False'; ExternalWritable := 'False'; } AT MyWord : Array[0..1] of Byte;
      MyBoolsinWord { ExternalAccessible := 'False'; ExternalVisible := 'False'; ExternalWritable := 'False'; } AT MyWord : Array[0..15] of Bool;
      MyDInt { ExternalAccessible := 'False'; ExternalVisible := 'False'; ExternalWritable := 'False'; } : DInt;
      MyWordsinDint { ExternalAccessible := 'False'; ExternalVisible := 'False'; ExternalWritable := 'False'; } AT MyDInt : Array[0..1] of Word;
      MyReal { ExternalAccessible := 'False'; ExternalVisible := 'False'; ExternalWritable := 'False'; } : Real;
      MyWordsinReal { ExternalAccessible := 'False'; ExternalVisible := 'False'; ExternalWritable := 'False'; } AT MyReal : Array[0..1] of Word;
      MyInt { ExternalAccessible := 'False'; ExternalVisible := 'False'; ExternalWritable := 'False'; } : Int;
      MyWordinInt { ExternalAccessible := 'False'; ExternalVisible := 'False'; ExternalWritable := 'False'; } AT MyInt : Word;
      MyDWord { ExternalAccessible := 'False'; ExternalVisible := 'False'; ExternalWritable := 'False'; } : DWord;
      MyWordsinDWord { ExternalAccessible := 'False'; ExternalVisible := 'False'; ExternalWritable := 'False'; } AT MyDWord : Array[0..1] of Word;
      MyTime { ExternalAccessible := 'False'; ExternalVisible := 'False'; ExternalWritable := 'False'; } : Time;
      MyWordsinTime { ExternalAccessible := 'False'; ExternalVisible := 'False'; ExternalWritable := 'False'; } AT MyTime : Array[0..1] of Word;
      MyString { ExternalAccessible := 'False'; ExternalVisible := 'False'; ExternalWritable := 'False'; } : String[40];
      MyWordsinString { ExternalAccessible := 'False'; ExternalVisible := 'False'; ExternalWritable := 'False'; } AT MyString : Array[0..20] of Word;
   END_VAR
   VAR_TEMP
      HashModbus : DInt;
      HashIFA : DInt;
      HashTIAMap : DInt;
      i : Int;
   END_VAR
    //Author: Miklos Boros (miklos.boros@esss.se), Copyrigth 2017-2019 by European Spallation Source, Lund
    //This block was generated by PLCFactory, please don't change it MANUALLY!
    //Input File Name: ISrc-010_Ctrl-PLC-01-template-IFA-20191106135317.ifa
    //Generated: 20191106135317
    //According to HASH: 1347332123
    //Device type: ISRC_LEBT_HVPS
    //Description: This function does the variable mapping for a device. All device-variable will be linked to an interface variable defined in this block.

    //********************************************
    //****************HASH check******************
    //********************************************


    #MyWordsinDint[0] := "EPICSToPLC"."Word"[0];
    #MyWordsinDint[1] := "EPICSToPLC"."Word"[1];
    #HashModbus := #MyDInt; //Hash from EPICS/ModbusTCP

    #HashIFA := 1347332123; //Hash from Interface Factory as a constant

    #MyWordsinDint[0] := "PLCToEPICS"."Word"[0];
    #MyWordsinDint[1] := "PLCToEPICS"."Word"[1];
    #HashTIAMap := #MyDInt; //Hash from PLCFactory TIA Map


    IF ((#HashIFA = #HashModbus) AND (#HashModbus = #HashTIAMap)) THEN //Check CRCs
        #DEVICE_PARAM_OK := TRUE;
       //###########################  ISrc HVPS  ##############################
       //###########################
       //STATUS BLOCK
       //###########################

    //********************************************
    //*************STATUS VARIABLES***************
    //********************************************


       #MyWord := W#0;
       #MyBoolsinWord[8] := #"ITLckEnCmdR";    //EPICSName: ITLckEnCmdR
       #MyBoolsinWord[9] := #"HVPSVolOK_Magtr";    //EPICSName: HVPSVolOK_Magtr
       "PLCToEPICS"."Word"[#PLCToEPICSDataBlockOffset + 0] := #MyWord;

    //********************************************
    //*************COMMAND VARIABLES**************
    //********************************************


       #MyWord := "EPICSToPLC"."Word"[#EPICSToPLCDataBlockOffset + 0];
       IF (NOT "Utilities".TestInProgress) THEN
       	"EPICSToPLC"."Word"[#EPICSToPLCDataBlockOffset + 0] := 0;
       END_IF;
       #"ESTOP" := #MyBoolsinWord[8];    //EPICSName: ESTOP

    //********************************************
    //************PARAMETER VARIABLES*************
    //********************************************


       #MyReal	:= 0.0;
       #MyWordsinReal[0]	:= "EPICSToPLC"."Word"[#EPICSToPLCDataBlockOffset + 1];
       #MyWordsinReal[1]	:= "EPICSToPLC"."Word"[#EPICSToPLCDataBlockOffset + 2];
       #"iVolR" := #MyReal;    //EPICSName: iVolR

       #MyWord := "EPICSToPLC"."Word"[#EPICSToPLCDataBlockOffset + 3];
       #"EPICSConnErr" := #MyBoolsinWord[8];    //EPICSName: EPICSConnErr
    Else
       #DEVICE_PARAM_OK := FALSE; //Invalid Hash
    END_IF;
END_FUNCTION_BLOCK
FUNCTION_BLOCK "DEVTYPE_ISRC_LEBT_HVPf_Doors"
{ S7_Optimized_Access := 'TRUE' }
VERSION : 1.0
   VAR_INPUT
      "CloseR" { ExternalAccessible := 'True'; ExternalVisible := 'False'; ExternalWritable := 'False'; } : BOOL;   //EPICS Status variable: CloseR
   EPICSToPLCLength { ExternalAccessible := 'False'; ExternalVisible := 'False'; ExternalWritable := 'False'; } : Int;   // Length of device command register array (in words)
   EPICSToPLCDataBlockOffset { ExternalAccessible := 'False'; ExternalVisible := 'False'; ExternalWritable := 'False'; } : Int;   // Offset in EPICS->PLC comms block where this device data resides (in words)
   EPICSToPLCParametersStart { ExternalAccessible := 'False'; ExternalVisible := 'False'; ExternalWritable := 'False'; } : Int;   // The border offset between the Command and the Parameter area
   PLCToEPICSLength { ExternalAccessible := 'False'; ExternalVisible := 'False'; ExternalWritable := 'False'; } : Int;   // Length of device status register array (in words)
   PLCToEPICSDataBlockOffset { ExternalAccessible := 'False'; ExternalVisible := 'False'; ExternalWritable := 'False'; } : Int;   // Offset in PLC->EPICS comms block where this device data resides (in words)
   END_VAR
   VAR_OUTPUT
      DEVICE_PARAM_OK { ExternalAccessible := 'False'; ExternalVisible := 'False'; ExternalWritable := 'False'; } : Bool;
   END_VAR
   VAR_IN_OUT
   END_VAR
   Var DB_SPECIFIC
      MyWord { ExternalAccessible := 'False'; ExternalVisible := 'False'; ExternalWritable := 'False'; } : Word;
      MyBytesinWord { ExternalAccessible := 'False'; ExternalVisible := 'False'; ExternalWritable := 'False'; } AT MyWord : Array[0..1] of Byte;
      MyBoolsinWord { ExternalAccessible := 'False'; ExternalVisible := 'False'; ExternalWritable := 'False'; } AT MyWord : Array[0..15] of Bool;
      MyDInt { ExternalAccessible := 'False'; ExternalVisible := 'False'; ExternalWritable := 'False'; } : DInt;
      MyWordsinDint { ExternalAccessible := 'False'; ExternalVisible := 'False'; ExternalWritable := 'False'; } AT MyDInt : Array[0..1] of Word;
      MyReal { ExternalAccessible := 'False'; ExternalVisible := 'False'; ExternalWritable := 'False'; } : Real;
      MyWordsinReal { ExternalAccessible := 'False'; ExternalVisible := 'False'; ExternalWritable := 'False'; } AT MyReal : Array[0..1] of Word;
      MyInt { ExternalAccessible := 'False'; ExternalVisible := 'False'; ExternalWritable := 'False'; } : Int;
      MyWordinInt { ExternalAccessible := 'False'; ExternalVisible := 'False'; ExternalWritable := 'False'; } AT MyInt : Word;
      MyDWord { ExternalAccessible := 'False'; ExternalVisible := 'False'; ExternalWritable := 'False'; } : DWord;
      MyWordsinDWord { ExternalAccessible := 'False'; ExternalVisible := 'False'; ExternalWritable := 'False'; } AT MyDWord : Array[0..1] of Word;
      MyTime { ExternalAccessible := 'False'; ExternalVisible := 'False'; ExternalWritable := 'False'; } : Time;
      MyWordsinTime { ExternalAccessible := 'False'; ExternalVisible := 'False'; ExternalWritable := 'False'; } AT MyTime : Array[0..1] of Word;
      MyString { ExternalAccessible := 'False'; ExternalVisible := 'False'; ExternalWritable := 'False'; } : String[40];
      MyWordsinString { ExternalAccessible := 'False'; ExternalVisible := 'False'; ExternalWritable := 'False'; } AT MyString : Array[0..20] of Word;
   END_VAR
   VAR_TEMP
      HashModbus : DInt;
      HashIFA : DInt;
      HashTIAMap : DInt;
      i : Int;
   END_VAR
    //Author: Miklos Boros (miklos.boros@esss.se), Copyrigth 2017-2019 by European Spallation Source, Lund
    //This block was generated by PLCFactory, please don't change it MANUALLY!
    //Input File Name: ISrc-010_Ctrl-PLC-01-template-IFA-20191106135317.ifa
    //Generated: 20191106135317
    //According to HASH: 1347332123
    //Device type: ISRC_LEBT_HVPf_Doors
    //Description: This function does the variable mapping for a device. All device-variable will be linked to an interface variable defined in this block.

    //********************************************
    //****************HASH check******************
    //********************************************


    #MyWordsinDint[0] := "EPICSToPLC"."Word"[0];
    #MyWordsinDint[1] := "EPICSToPLC"."Word"[1];
    #HashModbus := #MyDInt; //Hash from EPICS/ModbusTCP

    #HashIFA := 1347332123; //Hash from Interface Factory as a constant

    #MyWordsinDint[0] := "PLCToEPICS"."Word"[0];
    #MyWordsinDint[1] := "PLCToEPICS"."Word"[1];
    #HashTIAMap := #MyDInt; //Hash from PLCFactory TIA Map


    IF ((#HashIFA = #HashModbus) AND (#HashModbus = #HashTIAMap)) THEN //Check CRCs
        #DEVICE_PARAM_OK := TRUE;
       //#############################  ISRC HVPf Doors Status ##############################
       //###########################
       //STATUS BLOCK
       //###########################

    //********************************************
    //*************STATUS VARIABLES***************
    //********************************************


       #MyWord := W#0;
       #MyBoolsinWord[8] := #"CloseR";    //EPICSName: CloseR
       "PLCToEPICS"."Word"[#PLCToEPICSDataBlockOffset + 0] := #MyWord;
    Else
       #DEVICE_PARAM_OK := FALSE; //Invalid Hash
    END_IF;
END_FUNCTION_BLOCK
FUNCTION_BLOCK "DEVTYPE_ISRC_LEBT_HVPf_Res"
{ S7_Optimized_Access := 'TRUE' }
VERSION : 1.0
   VAR_INPUT
      "CloseR" { ExternalAccessible := 'True'; ExternalVisible := 'False'; ExternalWritable := 'False'; } : BOOL;   //EPICS Status variable: CloseR
   EPICSToPLCLength { ExternalAccessible := 'False'; ExternalVisible := 'False'; ExternalWritable := 'False'; } : Int;   // Length of device command register array (in words)
   EPICSToPLCDataBlockOffset { ExternalAccessible := 'False'; ExternalVisible := 'False'; ExternalWritable := 'False'; } : Int;   // Offset in EPICS->PLC comms block where this device data resides (in words)
   EPICSToPLCParametersStart { ExternalAccessible := 'False'; ExternalVisible := 'False'; ExternalWritable := 'False'; } : Int;   // The border offset between the Command and the Parameter area
   PLCToEPICSLength { ExternalAccessible := 'False'; ExternalVisible := 'False'; ExternalWritable := 'False'; } : Int;   // Length of device status register array (in words)
   PLCToEPICSDataBlockOffset { ExternalAccessible := 'False'; ExternalVisible := 'False'; ExternalWritable := 'False'; } : Int;   // Offset in PLC->EPICS comms block where this device data resides (in words)
   END_VAR
   VAR_OUTPUT
      DEVICE_PARAM_OK { ExternalAccessible := 'False'; ExternalVisible := 'False'; ExternalWritable := 'False'; } : Bool;
   END_VAR
   VAR_IN_OUT
   END_VAR
   Var DB_SPECIFIC
      MyWord { ExternalAccessible := 'False'; ExternalVisible := 'False'; ExternalWritable := 'False'; } : Word;
      MyBytesinWord { ExternalAccessible := 'False'; ExternalVisible := 'False'; ExternalWritable := 'False'; } AT MyWord : Array[0..1] of Byte;
      MyBoolsinWord { ExternalAccessible := 'False'; ExternalVisible := 'False'; ExternalWritable := 'False'; } AT MyWord : Array[0..15] of Bool;
      MyDInt { ExternalAccessible := 'False'; ExternalVisible := 'False'; ExternalWritable := 'False'; } : DInt;
      MyWordsinDint { ExternalAccessible := 'False'; ExternalVisible := 'False'; ExternalWritable := 'False'; } AT MyDInt : Array[0..1] of Word;
      MyReal { ExternalAccessible := 'False'; ExternalVisible := 'False'; ExternalWritable := 'False'; } : Real;
      MyWordsinReal { ExternalAccessible := 'False'; ExternalVisible := 'False'; ExternalWritable := 'False'; } AT MyReal : Array[0..1] of Word;
      MyInt { ExternalAccessible := 'False'; ExternalVisible := 'False'; ExternalWritable := 'False'; } : Int;
      MyWordinInt { ExternalAccessible := 'False'; ExternalVisible := 'False'; ExternalWritable := 'False'; } AT MyInt : Word;
      MyDWord { ExternalAccessible := 'False'; ExternalVisible := 'False'; ExternalWritable := 'False'; } : DWord;
      MyWordsinDWord { ExternalAccessible := 'False'; ExternalVisible := 'False'; ExternalWritable := 'False'; } AT MyDWord : Array[0..1] of Word;
      MyTime { ExternalAccessible := 'False'; ExternalVisible := 'False'; ExternalWritable := 'False'; } : Time;
      MyWordsinTime { ExternalAccessible := 'False'; ExternalVisible := 'False'; ExternalWritable := 'False'; } AT MyTime : Array[0..1] of Word;
      MyString { ExternalAccessible := 'False'; ExternalVisible := 'False'; ExternalWritable := 'False'; } : String[40];
      MyWordsinString { ExternalAccessible := 'False'; ExternalVisible := 'False'; ExternalWritable := 'False'; } AT MyString : Array[0..20] of Word;
   END_VAR
   VAR_TEMP
      HashModbus : DInt;
      HashIFA : DInt;
      HashTIAMap : DInt;
      i : Int;
   END_VAR
    //Author: Miklos Boros (miklos.boros@esss.se), Copyrigth 2017-2019 by European Spallation Source, Lund
    //This block was generated by PLCFactory, please don't change it MANUALLY!
    //Input File Name: ISrc-010_Ctrl-PLC-01-template-IFA-20191106135317.ifa
    //Generated: 20191106135317
    //According to HASH: 1347332123
    //Device type: ISRC_LEBT_HVPf_Res
    //Description: This function does the variable mapping for a device. All device-variable will be linked to an interface variable defined in this block.

    //********************************************
    //****************HASH check******************
    //********************************************


    #MyWordsinDint[0] := "EPICSToPLC"."Word"[0];
    #MyWordsinDint[1] := "EPICSToPLC"."Word"[1];
    #HashModbus := #MyDInt; //Hash from EPICS/ModbusTCP

    #HashIFA := 1347332123; //Hash from Interface Factory as a constant

    #MyWordsinDint[0] := "PLCToEPICS"."Word"[0];
    #MyWordsinDint[1] := "PLCToEPICS"."Word"[1];
    #HashTIAMap := #MyDInt; //Hash from PLCFactory TIA Map


    IF ((#HashIFA = #HashModbus) AND (#HashModbus = #HashTIAMap)) THEN //Check CRCs
        #DEVICE_PARAM_OK := TRUE;
       //###########################  HVPf Neutral To Ground Resistor Switches  ##############################
       //###########################
       //STATUS BLOCK
       //###########################

    //********************************************
    //*************STATUS VARIABLES***************
    //********************************************


       #MyWord := W#0;
       #MyBoolsinWord[8] := #"CloseR";    //EPICSName: CloseR
       "PLCToEPICS"."Word"[#PLCToEPICSDataBlockOffset + 0] := #MyWord;
    Else
       #DEVICE_PARAM_OK := FALSE; //Invalid Hash
    END_IF;
END_FUNCTION_BLOCK
FUNCTION_BLOCK "DEVTYPE_ISRC_LEBT_INTF_DIAG"
{ S7_Optimized_Access := 'TRUE' }
VERSION : 1.0
   VAR_INPUT
      "CPU_Connected" { ExternalAccessible := 'True'; ExternalVisible := 'False'; ExternalWritable := 'False'; } : BOOL;   //EPICS Status variable: CPU_Connected
      "DI1_Connected" { ExternalAccessible := 'True'; ExternalVisible := 'False'; ExternalWritable := 'False'; } : BOOL;   //EPICS Status variable: DI1_Connected
      "DI2_Connected" { ExternalAccessible := 'True'; ExternalVisible := 'False'; ExternalWritable := 'False'; } : BOOL;   //EPICS Status variable: DI2_Connected
      "AI1_Connected" { ExternalAccessible := 'True'; ExternalVisible := 'False'; ExternalWritable := 'False'; } : BOOL;   //EPICS Status variable: AI1_Connected
      "AI2_Connected" { ExternalAccessible := 'True'; ExternalVisible := 'False'; ExternalWritable := 'False'; } : BOOL;   //EPICS Status variable: AI2_Connected
      "DO1_Connected" { ExternalAccessible := 'True'; ExternalVisible := 'False'; ExternalWritable := 'False'; } : BOOL;   //EPICS Status variable: DO1_Connected
      "DO2_Connected" { ExternalAccessible := 'True'; ExternalVisible := 'False'; ExternalWritable := 'False'; } : BOOL;   //EPICS Status variable: DO2_Connected
      "CPU_Status" { ExternalAccessible := 'True'; ExternalVisible := 'False'; ExternalWritable := 'False'; } : BOOL;   //EPICS Status variable: CPU_Status
      "DI1_Status" { ExternalAccessible := 'True'; ExternalVisible := 'False'; ExternalWritable := 'False'; } : BOOL;   //EPICS Status variable: DI1_Status
      "DI2_Status" { ExternalAccessible := 'True'; ExternalVisible := 'False'; ExternalWritable := 'False'; } : BOOL;   //EPICS Status variable: DI2_Status
      "AI1_Status" { ExternalAccessible := 'True'; ExternalVisible := 'False'; ExternalWritable := 'False'; } : BOOL;   //EPICS Status variable: AI1_Status
      "AI2_Status" { ExternalAccessible := 'True'; ExternalVisible := 'False'; ExternalWritable := 'False'; } : BOOL;   //EPICS Status variable: AI2_Status
      "DO1_Status" { ExternalAccessible := 'True'; ExternalVisible := 'False'; ExternalWritable := 'False'; } : BOOL;   //EPICS Status variable: DO1_Status
      "DO2_Status" { ExternalAccessible := 'True'; ExternalVisible := 'False'; ExternalWritable := 'False'; } : BOOL;   //EPICS Status variable: DO2_Status
      "RIO_Connected" { ExternalAccessible := 'True'; ExternalVisible := 'False'; ExternalWritable := 'False'; } : BOOL;   //EPICS Status variable: RIO_Connected
      "RIO_DI1_Connected" { ExternalAccessible := 'True'; ExternalVisible := 'False'; ExternalWritable := 'False'; } : BOOL;   //EPICS Status variable: RIO_DI1_Connected
      "RIO_DI2_Connected" { ExternalAccessible := 'True'; ExternalVisible := 'False'; ExternalWritable := 'False'; } : BOOL;   //EPICS Status variable: RIO_DI2_Connected
      "RIO_AI1_Connected" { ExternalAccessible := 'True'; ExternalVisible := 'False'; ExternalWritable := 'False'; } : BOOL;   //EPICS Status variable: RIO_AI1_Connected
      "RIO_DO1_Connected" { ExternalAccessible := 'True'; ExternalVisible := 'False'; ExternalWritable := 'False'; } : BOOL;   //EPICS Status variable: RIO_DO1_Connected
      "RIO_Status" { ExternalAccessible := 'True'; ExternalVisible := 'False'; ExternalWritable := 'False'; } : BOOL;   //EPICS Status variable: RIO_Status
      "RIO_DI1_Status" { ExternalAccessible := 'True'; ExternalVisible := 'False'; ExternalWritable := 'False'; } : BOOL;   //EPICS Status variable: RIO_DI1_Status
      "RIO_DI2_Status" { ExternalAccessible := 'True'; ExternalVisible := 'False'; ExternalWritable := 'False'; } : BOOL;   //EPICS Status variable: RIO_DI2_Status
      "RIO_AI1_Status" { ExternalAccessible := 'True'; ExternalVisible := 'False'; ExternalWritable := 'False'; } : BOOL;   //EPICS Status variable: RIO_AI1_Status
      "RIO_DO1_Status" { ExternalAccessible := 'True'; ExternalVisible := 'False'; ExternalWritable := 'False'; } : BOOL;   //EPICS Status variable: RIO_DO1_Status
   EPICSToPLCLength { ExternalAccessible := 'False'; ExternalVisible := 'False'; ExternalWritable := 'False'; } : Int;   // Length of device command register array (in words)
   EPICSToPLCDataBlockOffset { ExternalAccessible := 'False'; ExternalVisible := 'False'; ExternalWritable := 'False'; } : Int;   // Offset in EPICS->PLC comms block where this device data resides (in words)
   EPICSToPLCParametersStart { ExternalAccessible := 'False'; ExternalVisible := 'False'; ExternalWritable := 'False'; } : Int;   // The border offset between the Command and the Parameter area
   PLCToEPICSLength { ExternalAccessible := 'False'; ExternalVisible := 'False'; ExternalWritable := 'False'; } : Int;   // Length of device status register array (in words)
   PLCToEPICSDataBlockOffset { ExternalAccessible := 'False'; ExternalVisible := 'False'; ExternalWritable := 'False'; } : Int;   // Offset in PLC->EPICS comms block where this device data resides (in words)
   END_VAR
   VAR_OUTPUT
      DEVICE_PARAM_OK { ExternalAccessible := 'False'; ExternalVisible := 'False'; ExternalWritable := 'False'; } : Bool;
   END_VAR
   VAR_IN_OUT
   END_VAR
   Var DB_SPECIFIC
      MyWord { ExternalAccessible := 'False'; ExternalVisible := 'False'; ExternalWritable := 'False'; } : Word;
      MyBytesinWord { ExternalAccessible := 'False'; ExternalVisible := 'False'; ExternalWritable := 'False'; } AT MyWord : Array[0..1] of Byte;
      MyBoolsinWord { ExternalAccessible := 'False'; ExternalVisible := 'False'; ExternalWritable := 'False'; } AT MyWord : Array[0..15] of Bool;
      MyDInt { ExternalAccessible := 'False'; ExternalVisible := 'False'; ExternalWritable := 'False'; } : DInt;
      MyWordsinDint { ExternalAccessible := 'False'; ExternalVisible := 'False'; ExternalWritable := 'False'; } AT MyDInt : Array[0..1] of Word;
      MyReal { ExternalAccessible := 'False'; ExternalVisible := 'False'; ExternalWritable := 'False'; } : Real;
      MyWordsinReal { ExternalAccessible := 'False'; ExternalVisible := 'False'; ExternalWritable := 'False'; } AT MyReal : Array[0..1] of Word;
      MyInt { ExternalAccessible := 'False'; ExternalVisible := 'False'; ExternalWritable := 'False'; } : Int;
      MyWordinInt { ExternalAccessible := 'False'; ExternalVisible := 'False'; ExternalWritable := 'False'; } AT MyInt : Word;
      MyDWord { ExternalAccessible := 'False'; ExternalVisible := 'False'; ExternalWritable := 'False'; } : DWord;
      MyWordsinDWord { ExternalAccessible := 'False'; ExternalVisible := 'False'; ExternalWritable := 'False'; } AT MyDWord : Array[0..1] of Word;
      MyTime { ExternalAccessible := 'False'; ExternalVisible := 'False'; ExternalWritable := 'False'; } : Time;
      MyWordsinTime { ExternalAccessible := 'False'; ExternalVisible := 'False'; ExternalWritable := 'False'; } AT MyTime : Array[0..1] of Word;
      MyString { ExternalAccessible := 'False'; ExternalVisible := 'False'; ExternalWritable := 'False'; } : String[40];
      MyWordsinString { ExternalAccessible := 'False'; ExternalVisible := 'False'; ExternalWritable := 'False'; } AT MyString : Array[0..20] of Word;
   END_VAR
   VAR_TEMP
      HashModbus : DInt;
      HashIFA : DInt;
      HashTIAMap : DInt;
      i : Int;
   END_VAR
    //Author: Miklos Boros (miklos.boros@esss.se), Copyrigth 2017-2019 by European Spallation Source, Lund
    //This block was generated by PLCFactory, please don't change it MANUALLY!
    //Input File Name: ISrc-010_Ctrl-PLC-01-template-IFA-20191106135317.ifa
    //Generated: 20191106135317
    //According to HASH: 1347332123
    //Device type: ISRC_LEBT_INTF_DIAG
    //Description: This function does the variable mapping for a device. All device-variable will be linked to an interface variable defined in this block.

    //********************************************
    //****************HASH check******************
    //********************************************


    #MyWordsinDint[0] := "EPICSToPLC"."Word"[0];
    #MyWordsinDint[1] := "EPICSToPLC"."Word"[1];
    #HashModbus := #MyDInt; //Hash from EPICS/ModbusTCP

    #HashIFA := 1347332123; //Hash from Interface Factory as a constant

    #MyWordsinDint[0] := "PLCToEPICS"."Word"[0];
    #MyWordsinDint[1] := "PLCToEPICS"."Word"[1];
    #HashTIAMap := #MyDInt; //Hash from PLCFactory TIA Map


    IF ((#HashIFA = #HashModbus) AND (#HashModbus = #HashTIAMap)) THEN //Check CRCs
        #DEVICE_PARAM_OK := TRUE;
       //###########################  ISRC PLC Diagnostics  ##############################
       //###########################
       //STATUS BLOCK
       //###########################
       //Local modules connection state

    //********************************************
    //*************STATUS VARIABLES***************
    //********************************************


       #MyWord := W#0;
       #MyBoolsinWord[8] := #"CPU_Connected";    //EPICSName: CPU_Connected
       #MyBoolsinWord[9] := #"DI1_Connected";    //EPICSName: DI1_Connected
       #MyBoolsinWord[10] := #"DI2_Connected";    //EPICSName: DI2_Connected
       #MyBoolsinWord[11] := #"AI1_Connected";    //EPICSName: AI1_Connected
       #MyBoolsinWord[12] := #"AI2_Connected";    //EPICSName: AI2_Connected
       #MyBoolsinWord[13] := #"DO1_Connected";    //EPICSName: DO1_Connected
       #MyBoolsinWord[14] := #"DO2_Connected";    //EPICSName: DO2_Connected
       #MyBoolsinWord[15] := #"CPU_Status";    //EPICSName: CPU_Status
       #MyBoolsinWord[0] := #"DI1_Status";    //EPICSName: DI1_Status
       #MyBoolsinWord[1] := #"DI2_Status";    //EPICSName: DI2_Status
       #MyBoolsinWord[2] := #"AI1_Status";    //EPICSName: AI1_Status
       #MyBoolsinWord[3] := #"AI2_Status";    //EPICSName: AI2_Status
       #MyBoolsinWord[4] := #"DO1_Status";    //EPICSName: DO1_Status
       #MyBoolsinWord[5] := #"DO2_Status";    //EPICSName: DO2_Status
       #MyBoolsinWord[6] := #"RIO_Connected";    //EPICSName: RIO_Connected
       #MyBoolsinWord[7] := #"RIO_DI1_Connected";    //EPICSName: RIO_DI1_Connected
       "PLCToEPICS"."Word"[#PLCToEPICSDataBlockOffset + 0] := #MyWord;

       #MyWord := W#0;
       #MyBoolsinWord[8] := #"RIO_DI2_Connected";    //EPICSName: RIO_DI2_Connected
       #MyBoolsinWord[9] := #"RIO_AI1_Connected";    //EPICSName: RIO_AI1_Connected
       #MyBoolsinWord[10] := #"RIO_DO1_Connected";    //EPICSName: RIO_DO1_Connected
       #MyBoolsinWord[11] := #"RIO_Status";    //EPICSName: RIO_Status
       #MyBoolsinWord[12] := #"RIO_DI1_Status";    //EPICSName: RIO_DI1_Status
       #MyBoolsinWord[13] := #"RIO_DI2_Status";    //EPICSName: RIO_DI2_Status
       #MyBoolsinWord[14] := #"RIO_AI1_Status";    //EPICSName: RIO_AI1_Status
       #MyBoolsinWord[15] := #"RIO_DO1_Status";    //EPICSName: RIO_DO1_Status
       "PLCToEPICS"."Word"[#PLCToEPICSDataBlockOffset + 1] := #MyWord;
    Else
       #DEVICE_PARAM_OK := FALSE; //Invalid Hash
    END_IF;
END_FUNCTION_BLOCK
FUNCTION_BLOCK "DEVTYPE_ISRC_LEBT_INTF_DPL"
{ S7_Optimized_Access := 'TRUE' }
VERSION : 1.0
   VAR_INPUT
      "DPLOK" { ExternalAccessible := 'True'; ExternalVisible := 'False'; ExternalWritable := 'False'; } : BOOL;   //EPICS Status variable: DPLOK
   EPICSToPLCLength { ExternalAccessible := 'False'; ExternalVisible := 'False'; ExternalWritable := 'False'; } : Int;   // Length of device command register array (in words)
   EPICSToPLCDataBlockOffset { ExternalAccessible := 'False'; ExternalVisible := 'False'; ExternalWritable := 'False'; } : Int;   // Offset in EPICS->PLC comms block where this device data resides (in words)
   EPICSToPLCParametersStart { ExternalAccessible := 'False'; ExternalVisible := 'False'; ExternalWritable := 'False'; } : Int;   // The border offset between the Command and the Parameter area
   PLCToEPICSLength { ExternalAccessible := 'False'; ExternalVisible := 'False'; ExternalWritable := 'False'; } : Int;   // Length of device status register array (in words)
   PLCToEPICSDataBlockOffset { ExternalAccessible := 'False'; ExternalVisible := 'False'; ExternalWritable := 'False'; } : Int;   // Offset in PLC->EPICS comms block where this device data resides (in words)
   END_VAR
   VAR_OUTPUT
      DEVICE_PARAM_OK { ExternalAccessible := 'False'; ExternalVisible := 'False'; ExternalWritable := 'False'; } : Bool;
   END_VAR
   VAR_IN_OUT
   END_VAR
   Var DB_SPECIFIC
      MyWord { ExternalAccessible := 'False'; ExternalVisible := 'False'; ExternalWritable := 'False'; } : Word;
      MyBytesinWord { ExternalAccessible := 'False'; ExternalVisible := 'False'; ExternalWritable := 'False'; } AT MyWord : Array[0..1] of Byte;
      MyBoolsinWord { ExternalAccessible := 'False'; ExternalVisible := 'False'; ExternalWritable := 'False'; } AT MyWord : Array[0..15] of Bool;
      MyDInt { ExternalAccessible := 'False'; ExternalVisible := 'False'; ExternalWritable := 'False'; } : DInt;
      MyWordsinDint { ExternalAccessible := 'False'; ExternalVisible := 'False'; ExternalWritable := 'False'; } AT MyDInt : Array[0..1] of Word;
      MyReal { ExternalAccessible := 'False'; ExternalVisible := 'False'; ExternalWritable := 'False'; } : Real;
      MyWordsinReal { ExternalAccessible := 'False'; ExternalVisible := 'False'; ExternalWritable := 'False'; } AT MyReal : Array[0..1] of Word;
      MyInt { ExternalAccessible := 'False'; ExternalVisible := 'False'; ExternalWritable := 'False'; } : Int;
      MyWordinInt { ExternalAccessible := 'False'; ExternalVisible := 'False'; ExternalWritable := 'False'; } AT MyInt : Word;
      MyDWord { ExternalAccessible := 'False'; ExternalVisible := 'False'; ExternalWritable := 'False'; } : DWord;
      MyWordsinDWord { ExternalAccessible := 'False'; ExternalVisible := 'False'; ExternalWritable := 'False'; } AT MyDWord : Array[0..1] of Word;
      MyTime { ExternalAccessible := 'False'; ExternalVisible := 'False'; ExternalWritable := 'False'; } : Time;
      MyWordsinTime { ExternalAccessible := 'False'; ExternalVisible := 'False'; ExternalWritable := 'False'; } AT MyTime : Array[0..1] of Word;
      MyString { ExternalAccessible := 'False'; ExternalVisible := 'False'; ExternalWritable := 'False'; } : String[40];
      MyWordsinString { ExternalAccessible := 'False'; ExternalVisible := 'False'; ExternalWritable := 'False'; } AT MyString : Array[0..20] of Word;
   END_VAR
   VAR_TEMP
      HashModbus : DInt;
      HashIFA : DInt;
      HashTIAMap : DInt;
      i : Int;
   END_VAR
    //Author: Miklos Boros (miklos.boros@esss.se), Copyrigth 2017-2019 by European Spallation Source, Lund
    //This block was generated by PLCFactory, please don't change it MANUALLY!
    //Input File Name: ISrc-010_Ctrl-PLC-01-template-IFA-20191106135317.ifa
    //Generated: 20191106135317
    //According to HASH: 1347332123
    //Device type: ISRC_LEBT_INTF_DPL
    //Description: This function does the variable mapping for a device. All device-variable will be linked to an interface variable defined in this block.

    //********************************************
    //****************HASH check******************
    //********************************************


    #MyWordsinDint[0] := "EPICSToPLC"."Word"[0];
    #MyWordsinDint[1] := "EPICSToPLC"."Word"[1];
    #HashModbus := #MyDInt; //Hash from EPICS/ModbusTCP

    #HashIFA := 1347332123; //Hash from Interface Factory as a constant

    #MyWordsinDint[0] := "PLCToEPICS"."Word"[0];
    #MyWordsinDint[1] := "PLCToEPICS"."Word"[1];
    #HashTIAMap := #MyDInt; //Hash from PLCFactory TIA Map


    IF ((#HashIFA = #HashModbus) AND (#HashModbus = #HashTIAMap)) THEN //Check CRCs
        #DEVICE_PARAM_OK := TRUE;
       //###########################  ISRC_LEBT interface with DPL  ##############################
       //###########################
       //STATUS BLOCK
       //###########################

    //********************************************
    //*************STATUS VARIABLES***************
    //********************************************


       #MyWord := W#0;
       #MyBoolsinWord[8] := #"DPLOK";    //EPICSName: DPLOK
       "PLCToEPICS"."Word"[#PLCToEPICSDataBlockOffset + 0] := #MyWord;
    Else
       #DEVICE_PARAM_OK := FALSE; //Invalid Hash
    END_IF;
END_FUNCTION_BLOCK
FUNCTION_BLOCK "DEVTYPE_ISRC_LEBT_INTF_EMU"
{ S7_Optimized_Access := 'TRUE' }
VERSION : 1.0
   VAR_INPUT
      "EMUOK" { ExternalAccessible := 'True'; ExternalVisible := 'False'; ExternalWritable := 'False'; } : BOOL;   //EPICS Status variable: EMUOK
      "EMUOK_Magtr" { ExternalAccessible := 'True'; ExternalVisible := 'False'; ExternalWritable := 'False'; } : BOOL;   //EPICS Status variable: EMUOK_Magtr
   EPICSToPLCLength { ExternalAccessible := 'False'; ExternalVisible := 'False'; ExternalWritable := 'False'; } : Int;   // Length of device command register array (in words)
   EPICSToPLCDataBlockOffset { ExternalAccessible := 'False'; ExternalVisible := 'False'; ExternalWritable := 'False'; } : Int;   // Offset in EPICS->PLC comms block where this device data resides (in words)
   EPICSToPLCParametersStart { ExternalAccessible := 'False'; ExternalVisible := 'False'; ExternalWritable := 'False'; } : Int;   // The border offset between the Command and the Parameter area
   PLCToEPICSLength { ExternalAccessible := 'False'; ExternalVisible := 'False'; ExternalWritable := 'False'; } : Int;   // Length of device status register array (in words)
   PLCToEPICSDataBlockOffset { ExternalAccessible := 'False'; ExternalVisible := 'False'; ExternalWritable := 'False'; } : Int;   // Offset in PLC->EPICS comms block where this device data resides (in words)
   END_VAR
   VAR_OUTPUT
      DEVICE_PARAM_OK { ExternalAccessible := 'False'; ExternalVisible := 'False'; ExternalWritable := 'False'; } : Bool;
   END_VAR
   VAR_IN_OUT
   END_VAR
   Var DB_SPECIFIC
      MyWord { ExternalAccessible := 'False'; ExternalVisible := 'False'; ExternalWritable := 'False'; } : Word;
      MyBytesinWord { ExternalAccessible := 'False'; ExternalVisible := 'False'; ExternalWritable := 'False'; } AT MyWord : Array[0..1] of Byte;
      MyBoolsinWord { ExternalAccessible := 'False'; ExternalVisible := 'False'; ExternalWritable := 'False'; } AT MyWord : Array[0..15] of Bool;
      MyDInt { ExternalAccessible := 'False'; ExternalVisible := 'False'; ExternalWritable := 'False'; } : DInt;
      MyWordsinDint { ExternalAccessible := 'False'; ExternalVisible := 'False'; ExternalWritable := 'False'; } AT MyDInt : Array[0..1] of Word;
      MyReal { ExternalAccessible := 'False'; ExternalVisible := 'False'; ExternalWritable := 'False'; } : Real;
      MyWordsinReal { ExternalAccessible := 'False'; ExternalVisible := 'False'; ExternalWritable := 'False'; } AT MyReal : Array[0..1] of Word;
      MyInt { ExternalAccessible := 'False'; ExternalVisible := 'False'; ExternalWritable := 'False'; } : Int;
      MyWordinInt { ExternalAccessible := 'False'; ExternalVisible := 'False'; ExternalWritable := 'False'; } AT MyInt : Word;
      MyDWord { ExternalAccessible := 'False'; ExternalVisible := 'False'; ExternalWritable := 'False'; } : DWord;
      MyWordsinDWord { ExternalAccessible := 'False'; ExternalVisible := 'False'; ExternalWritable := 'False'; } AT MyDWord : Array[0..1] of Word;
      MyTime { ExternalAccessible := 'False'; ExternalVisible := 'False'; ExternalWritable := 'False'; } : Time;
      MyWordsinTime { ExternalAccessible := 'False'; ExternalVisible := 'False'; ExternalWritable := 'False'; } AT MyTime : Array[0..1] of Word;
      MyString { ExternalAccessible := 'False'; ExternalVisible := 'False'; ExternalWritable := 'False'; } : String[40];
      MyWordsinString { ExternalAccessible := 'False'; ExternalVisible := 'False'; ExternalWritable := 'False'; } AT MyString : Array[0..20] of Word;
   END_VAR
   VAR_TEMP
      HashModbus : DInt;
      HashIFA : DInt;
      HashTIAMap : DInt;
      i : Int;
   END_VAR
    //Author: Miklos Boros (miklos.boros@esss.se), Copyrigth 2017-2019 by European Spallation Source, Lund
    //This block was generated by PLCFactory, please don't change it MANUALLY!
    //Input File Name: ISrc-010_Ctrl-PLC-01-template-IFA-20191106135317.ifa
    //Generated: 20191106135317
    //According to HASH: 1347332123
    //Device type: ISRC_LEBT_INTF_EMU
    //Description: This function does the variable mapping for a device. All device-variable will be linked to an interface variable defined in this block.

    //********************************************
    //****************HASH check******************
    //********************************************


    #MyWordsinDint[0] := "EPICSToPLC"."Word"[0];
    #MyWordsinDint[1] := "EPICSToPLC"."Word"[1];
    #HashModbus := #MyDInt; //Hash from EPICS/ModbusTCP

    #HashIFA := 1347332123; //Hash from Interface Factory as a constant

    #MyWordsinDint[0] := "PLCToEPICS"."Word"[0];
    #MyWordsinDint[1] := "PLCToEPICS"."Word"[1];
    #HashTIAMap := #MyDInt; //Hash from PLCFactory TIA Map


    IF ((#HashIFA = #HashModbus) AND (#HashModbus = #HashTIAMap)) THEN //Check CRCs
        #DEVICE_PARAM_OK := TRUE;
       //###########################  ISRC_LEBT interface with EMU  ##############################
       //###########################
       //STATUS BLOCK
       //###########################

    //********************************************
    //*************STATUS VARIABLES***************
    //********************************************


